// TIA Portal V17 export
// export: Created 2024-08-29T18:23:49.9514799Z, ExportSetting WithDefaults, DisplayName Totally Integrated Automation Portal, DisplayVersion V17 Update 7, DisplayName TIA Portal Openness, DisplayVersion V17 Update 7, DisplayName TIA Portal Version Control Interface, DisplayVersion V17, DisplayName SINAMICS Startdrive Advanced, DisplayVersion V17 SP2, DisplayName SINAMICS Startdrive G110M, G120, G120C, G120D, G120P, G115D, DisplayVersion V17 SP2, DisplayName SINAMICS Startdrive G130, G150, S120, S150, SINAMICS MV, S210, DisplayVersion V17 SP2, DisplayName STEP 7 Professional, DisplayVersion V17 Update 7, DisplayName STEP 7 Safety, DisplayVersion V17 Update 6, DisplayName WinCC Advanced / Unified PC, DisplayVersion V17 Update 7
VAR_GLOBAL   // PLC tag table "digitalFieldbusInputs"
   iRightTrackClampExt AT %I147.0 : Bool;
   iLeftTrackClampExt AT %I147.1 : Bool;
   iRightNestLocatingPinExt AT %I147.2 : Bool;
   iLeftNestLocatingPinExt AT %I147.3 : Bool;
   iRightTrackClampRet AT %I148.0 : Bool;
   iLeftTrackClampRet AT %I148.1 : Bool;
   iRightNestLocatingPinRet AT %I148.2 : Bool;
   iLeftNestLocatingPinRet AT %I148.3 : Bool;
   iLeftTrackPS1 AT %I149.0 : Bool;
   iLeftTrackPS2 AT %I149.1 : Bool;
   iRightTrackPS1 AT %I149.2 : Bool;
   iRightTrackPS2 AT %I149.3 : Bool;
   iLeftNestInitialPos AT %I149.4 : Bool;
   iRightNestInitialPos AT %I149.5 : Bool;
   iRightManualClampClosed AT %I149.6 : Bool;
   iLeftManualClampClosed AT %I149.7 : Bool;
   iPlasticBridgePS AT %I151.0 : Bool;
   iLeftNestWorkingPos AT %I151.1 : Bool;
   iPokayokeLeftTrackPS AT %I151.2 : Bool;
   iPokayokeRightTrackPS AT %I151.3 : Bool;
   iPlasticBridgeClampClosed AT %I151.4 : Bool;
   iInsertPlasticBridgePos AT %I151.6 : Bool;
   iInsertShaftPos AT %I151.7 : Bool;
END_VAR
